PROGRAM MAIN
VAR
	server_IntegrationTestSuite : Server_IntegrationTestSuite;
	chunkedRequestData_TestSuite : ChunkedRequestData_TestSuite;
	
	initialized : BOOL;
	server : RpcServer;
	concatStringRpcHandler : ConcatStringRpcHandler;	
	asyncEchoRpcHandler : AsyncEchoRpcHandler;
	adjustableSizeReplyRpcHandler : AdjustableSizeReplyRpcHandler;

END_VAR

TcUnit.RUN();

// the code below is used by TwinCAT HMI implementation

IF NOT initialized THEN
	initialized := TRUE;
	server.RegisterSynchronousRpcHandler('concat',concatStringRpcHandler);
	server.RegisterSynchronousRpcHandler('asyncEcho',asyncEchoRpcHandler);
	server.RegisterSynchronousRpcHandler('adjustableSizeReply',adjustableSizeReplyRpcHandler);
END_IF

server.CyclicCall();

// this has timers inside, so must be cyclic called.
asyncEchoRpcHandler.CyclicCall();

END_PROGRAM

(* stored: Version 1.1.0.1, ProductVersion 3.1.4024.12
   POU MAIN: Id {6a5ba616-dd43-4b8b-8788-947f674d5790}, SpecialFunc None *)
